FUNCTION_BLOCK EcMasterGetDeviceState IMPLEMENTS IEcTask
VAR_INPUT
END_VAR
VAR_OUTPUT
END_VAR
VAR
	iState : INT;
	getDeviceState : Tc2_EtherCAT.FB_EcGetSlaveState;
	_execute: BOOL;
	_done: BOOL;
	_busy: BOOL;
	_error: BOOL;
	_netId: AMSNETID;
END_VAR

CASE iState OF
	0:
		IF _execute THEN
			_done := FALSE;
			_busy := TRUE;
			_error := FALSE;
			getDeviceState.bExecute := TRUE;
			IF getDeviceState.bBusy THEN
				iState := 10;
				_execute := false;
			END_IF
		END_IF
	10:
		IF NOT getDeviceState.bBusy THEN
			IF NOT getDeviceState.bError THEN
				_done := TRUE;
			ELSE
				_error := TRUE;
			END_IF
			_busy := FALSE;
			getDeviceState.bExecute := FALSE;
			iState := 0;
		END_IF
END_CASE

getDeviceState(sNetId := Tc2_System.F_CreateAmsNetId(nIds := NetId));

{warning 'add method implementation '}
METHOD Abort : BOOL
getDeviceState.bExecute := FALSE;
_busy := FALSE;
_execute := FALSE;
Abort := TRUE;
iState := 0;
END_METHOD

{warning 'add property implementation'}
PROPERTY Busy : BOOL
GET
Busy := _busy;
END_GET
END_PROPERTY

PROPERTY DeviceAddr : uint
GET
DeviceAddr := getDeviceState.nSlaveAddr;
END_GET
SET
getDeviceState.nSlaveAddr := DeviceAddr;
END_SET
END_PROPERTY

PROPERTY DeviceState : ST_EcSlaveState
GET
DeviceState := getDeviceState.state;
END_GET
END_PROPERTY

{warning 'add property implementation'}
PROPERTY Done : BOOL
GET
Done := _done;
END_GET
END_PROPERTY

{warning 'add property implementation'}
PROPERTY Error : BOOL
GET
Error := _error;
END_GET
END_PROPERTY

{warning 'add method implementation '}
METHOD Execute : BOOL
IF NOT getDeviceState.bBusy THEN
	Execute := _execute := true;
END_IF
END_METHOD

{warning 'add property implementation'}
PROPERTY NetID : amsnetid
GET
NetID := _netId;
END_GET
SET
_netId := NetID;
END_SET
END_PROPERTY

END_FUNCTION_BLOCK

(* stored: Version 1.1.0.1, ProductVersion 3.1.4024.9
   POU EcMasterGetDeviceState: Id {8be47d8e-19f8-4ec1-a33d-cffdd276a9ac}, SpecialFunc None
   Method Abort: Id {24753508-e7b2-4fe3-83be-23d952dee1f9}
   Property Busy: Id {30f2df50-a0ce-413c-b8cc-4f53c64fb6cb}
   Get Get: Id {09cf52ca-abed-45d9-a657-1de9bad65b38}
   Property DeviceAddr: Id {5e495f62-e7ef-4658-9538-d28ec6916ee2}
   Get Get: Id {cf7c00d2-186b-495c-a03b-130707671078}
   Set Set: Id {a3d5a919-27b6-423c-888b-e4769e221f2e}
   Property DeviceState: Id {623750e0-7f94-48e0-9ce6-6ce0761a33e4}
   Get Get: Id {34644ede-8e9d-4452-af61-f39aa8a3cf91}
   Property Done: Id {e8a17d00-736a-413c-ae40-d511d62590de}
   Get Get: Id {ba462c4c-d7b3-45b5-9e9b-e7597c40667e}
   Property Error: Id {6025c8de-a9b8-4b98-be95-b2aefa1cf87e}
   Get Get: Id {71893dab-fcb8-4e37-96c2-b499efa7fe45}
   Method Execute: Id {8396ce43-feed-4def-ae1a-ffb894353886}
   Property NetID: Id {e08e0ff8-c1a9-47d4-98fd-27b652cc0dce}
   Get Get: Id {a3cc9c33-f26a-48c3-b07b-4e51aeeb78b3}
   Set Set: Id {7b96a686-175d-48b8-8400-7cb6ff85d0ab} *)
